FUNCTION_BLOCK MockEvent IMPLEMENTS I_Event
VAR
	_name : T_MAXSTRING;
END_VAR

METHOD FB_init : BOOL
VAR_INPUT
	bInitRetains : BOOL; // if TRUE, the retain variables are initialized (warm start / cold start)
	bInCopyCode : BOOL;  // if TRUE, the instance afterwards gets moved into the copy code (online change)
	Name : T_MAXSTRING;
END_VAR
_name := Name;
END_METHOD

PROPERTY Name : T_MaxString
GET
Name := _name;
END_GET
END_PROPERTY

END_FUNCTION_BLOCK

(* stored: Version 1.1.0.1, ProductVersion 3.1.4024.12
   POU MockEvent: Id {2f9c554a-2034-412e-9e68-a68075e23a21}, SpecialFunc None
   Folder Constructor: Id {92faa27c-d0c8-4754-92f3-0ceeacba4f84}
   Method FB_init: Id {db307f70-0de2-41b4-a82b-6e906a827d0e}
   Property Name: Id {bece4540-f580-49da-93aa-5dfe7c2b852d}
   Get Get: Id {72762b61-636c-4abe-8de9-0196d164a96e} *)
